// TwinCAT 3 PLC project Main
// ProgramVersion: 3.1.4023.0
// libraries:
//   mobject-collections, * (mobject)
//   mobject-enumerable, * (mobject)
//   mobject-events, * (mobject)
//   Tc2_System, * (Beckhoff Automation GmbH)
//   Tc3_Module, * (Beckhoff Automation GmbH)
//   TcUnit, * (www.tcunit.org)
// project tree:
//   / PlcTask.TcTTO
//   POUs/ Main.TcPOU
//   Tests/ OrderedDicKeyValueForwardEnumerator_TestSuite.TcPOU (not stored), OrderedDictionaryForwardEnumerator_TestSuite.TcPOU (not stored), DictionaryKeyValueForwardEnumerator_TestSuite.TcPOU (not stored), Dictionary_TestSuite.TcPOU (not stored), DictionaryForwardEnumerator_TestSuite.TcPOU (not stored), OrderedDictionary_TestSuite.TcPOU (not stored), LinkedList_TestSuite.TcPOU (not stored), ListForwardEnumerator_TestSuite.TcPOU, List_TestSuite.TcPOU, StackForwardEnumerator_TestSuite.TcPOU (not stored), Queue_TestSuite.TcPOU (not stored), LinkedListForwardEnumerator_TestSuite.TcPOU (not stored), Stack_TestSuite.TcPOU (not stored), QueueForwardEnumerator_TestSuite.TcPOU (not stored)
//   Tests/Mocks/EventHandlers/ CollectionChangedEventHandler.TcPOU (not stored), CollectionDisposedEventHandler.TcPOU (not stored), CollectionEventHandler.TcPOU (not stored), KeyValueCollectionChangedEventHandler.TcPOU (not stored), KeyValueCollectionEventHandler.TcPOU (not stored), KeyValueCollectionDisposedEventHandler.TcPOU (not stored), MockEventHandler.TcPOU (not stored)
// real-time tasks:
//   TASK PlcTask: cycle T#10ms, priority 20, ADS port 350

CONFIGURATION Main
    RESOURCE PLC ON TwinCAT3
        TASK PlcTask(INTERVAL := T#10ms, PRIORITY := 20);
        PROGRAM Main WITH PlcTask : Main;
    END_RESOURCE
END_CONFIGURATION

// ---- POUs/Main.TcPOU
PROGRAM Main
VAR
	dictionary_TestSuite : Dictionary_TestSuite;
	dictionaryForwardEnumerator_TestSuite : DictionaryForwardEnumerator_TestSuite;
	dictionaryKeyValueForwardEnumerator_TestSuite : DictionaryKeyValueForwardEnumerator_TestSuite;
	orderedDictionary_TestSuite : OrderedDictionary_TestSuite;
	orderedDictionaryForwardEnumerator_TestSuite : OrderedDictionaryForwardEnumerator_TestSuite;
	orderedDicKeyValueForwardEnumerator_TestSuite : OrderedDicKeyValueForwardEnumerator_TestSuite;
    linkedList_TestSuite : LinkedList_TestSuite;
	linkedListForwardEnumerator_TestSuite : LinkedListForwardEnumerator_TestSuite;
    list_TestSuite : List_TestSuite;
    listEnumerator_TestSuite : ListForwardEnumerator_TestSuite;
	queue_TestSuite : Queue_TestSuite;
	queueForwardEnumerator_TestSuite : QueueForwardEnumerator_TestSuite;
    stack_TestSuite : Stack_TestSuite;
	stackForwardEnumerator_TestSuite : StackForwardEnumerator_TestSuite;
END_VAR

TcUnit.Run();

END_PROGRAM

// ---- Tests/List_TestSuite.TcPOU
FUNCTION_BLOCK List_TestSuite EXTENDS TcUnit.FB_TestSuite
VAR
END_VAR

CheckAddItem();
CheckCapacityAfterAdding1Item();
CheckCapacityAfterAdding5Items();
CheckCapacityAfterAdding5ItemsTrimThen1Item();
CheckCapacityAtStart();
CheckClear();
CheckContains();
CheckTryCopyTo();
CheckTryCopyToLocation();
CheckCount();
CheckGetByIndexInBounds();
CheckGetByIndexNoItems();
CheckGetByIndexOutOfBounds();
CheckGetEnumerator();
CheckGetIndexOfExistingItem();
CheckGetIndexOfNonExistingItem();
CheckImplementsICollection();
CheckImplementsIList();
CheckTryInsert();
CheckOnChangedEvent();
CheckOnDisposedEvent();
CheckOnceEvent();
CheckOffEvent();
CheckTryRemoveAtInBounds();
CheckTryRemoveAtNoItems();
CheckTryRemoveAtOutOfBounds();
CheckTryRemoveItemFirstShiftUp();
CheckTryRemoveItemNonExisting();
CheckTryRemoveItemSecondShiftUp();
CheckTrimExcessAfterAdding5Items();
CheckIsEmptyWhenEmpty();
CheckIsEmptyWhenFull();

METHOD PRIVATE CheckAddItem
VAR
	in1 : INT := 123;
	in2 : INT := 456;
	in3 : INT := 789;
	out : INT;
	expected : INT := 789;
END_VAR
VAR_INST
	list : List;
END_VAR
TEST('CheckAddItem');

list.AddItem(in1); // [123]
list.AddItem(in2); // [123,456]
list.AddItem(in3); // [123,456,789]

list.TryGetByIndex(2, out);

AssertEquals(expected, out, 'Did not produce the expected result');

TEST_FINISHED();
END_METHOD

METHOD PRIVATE CheckCapacityAfterAdding1Item
VAR
	in1 : INT := 1;
	expected : DINT := 4;
	out : DINT;
END_VAR
VAR_INST
	list : List;
END_VAR
TEST('CheckCapacityAfterAdding1Item');

list.AddItem(in1); // [1, null, null, null]

out := list.Capacity;

AssertEquals(expected, out, 'List was expected to double once 5 items were added');

TEST_FINISHED();
END_METHOD

METHOD PRIVATE CheckCapacityAfterAdding5Items
VAR
	in1 : INT := 1;
	in2 : INT := 2;
	in3 : INT := 3;
	in4 : INT := 4;
	in5 : INT := 5;
	in6 : INT := 6;
	expected : DINT := 8;
	out : DINT;
END_VAR
VAR_INST
	list : List;
END_VAR
TEST('CheckCapacityAfterAdding5Items');

list.AddItem(in1); // [1, null, null, null]
list.AddItem(in2); // [1, 2, null, null]
list.AddItem(in3); // [1, 2, 3, null]
list.AddItem(in4); // [1, 2, 3, 4]
list.AddItem(in5); // [1, 2, 3, 4, 5, null, null, null]

out := list.Capacity;

AssertEquals(expected, out, 'List was expected to double once 5 items were added');

TEST_FINISHED();
END_METHOD

METHOD PRIVATE CheckCapacityAfterAdding5ItemsTrimThen1Item
VAR
	in1 : INT := 1;
	in2 : INT := 2;
	in3 : INT := 3;
	in4 : INT := 4;
	in5 : INT := 5;
	in6 : INT := 6;
	expected : DINT := 10;
	out : DINT;
END_VAR
VAR_INST
	list : List;
END_VAR
TEST('CheckCapacityAfterAdding5ItemsTrimThen1Item');

list.AddItem(in1); // [1, null, null, null]
list.AddItem(in2); // [1, 2, null, null]
list.AddItem(in3); // [1, 2, 3, null]
list.AddItem(in4); // [1, 2, 3, 4]
list.AddItem(in5); // [1, 2, 3, 4, 5, null, null, null]
list.TrimExcess(); // [1, 2, 3, 4, 5]
list.AddItem(in6); // [1, 2, 3, 4, 5, 6]

out := list.Capacity;

AssertEquals(expected, out, 'Incorrect capacity returned');

TEST_FINISHED();
END_METHOD

METHOD PRIVATE CheckCapacityAtStart
VAR
	expected : DINT := 0;
	out : DINT;
END_VAR
VAR_INST
	list : List;
END_VAR
TEST('CheckCapacityAtStart');

out := list.Capacity;

AssertEquals(expected, out, 'List was expected to start with a capacity of 0');

TEST_FINISHED();
END_METHOD

METHOD PRIVATE CheckClear
VAR
	in1 : INT := 123;
	in2 : INT := 456;
	in3 : INT := 789;
	expected : INT := 789;
	out : INT;
END_VAR
VAR_INST
	list : List;
END_VAR
TEST('CheckClear');

list.AddItem(in1); // [123]
list.AddItem(in2); // [123,456]

list.Clear(); // []
list.AddItem(in3); // [789]

list.TryGetByIndex(0, out);

AssertEquals(expected, out, 'Did not produce the expected result');

TEST_FINISHED();
END_METHOD

METHOD PRIVATE CheckContains
VAR
	in1 : INT := 123;
	in2 : INT := 456;
	in3 : INT := 789;
	result : BOOL;
END_VAR
VAR_INST
	list : List;
END_VAR
TEST('ListTests_CheckContains');

list.AddItem(in1); // [123]
list.AddItem(in2); // [123,456]
list.AddItem(in3); // [123,456,789]

result := list.Contains(in2);

AssertTrue(result, 'Contains returned false while item should be in collection');

TEST_FINISHED();
END_METHOD

METHOD PRIVATE CheckCount
VAR
	in1 : INT := 123;
	in2 : INT := 456;
	in3 : INT := 789;
	expected : DINT := 3;
	out : DINT;
END_VAR
VAR_INST
	list : List;
END_VAR
TEST('ListTests_CheckCount');

list.AddItem(in1); // [123]
list.AddItem(in2); // [123,456]
list.AddItem(in3); // [123,456,789]

out := list.Count;

AssertEquals(expected, out, 'Did not prodocue the expected result');

TEST_FINISHED();
END_METHOD

METHOD PRIVATE CheckGetByIndexInBounds
VAR
	in1 : INT := 123;
	in2 : INT := 456;
	in3 : INT := 789;
	out : INT;
	result : BOOL;
	expected : INT := 456;
END_VAR
VAR_INST
	list : List;
END_VAR
TEST('CheckGetByIndexInBounds');

list.AddItem(in1); // [123]
list.AddItem(in2); // [123,456]
list.AddItem(in3); // [123,456,789]

result := list.TryGetByIndex(1, out);

AssertTRUE(result, 'Returned FALSE while the index is populated');

AssertEquals(expected, out, 'Retrieved different value than expected');

TEST_FINISHED();
END_METHOD

METHOD PRIVATE CheckGetByIndexNoItems
VAR
	out : INT;
	result : BOOL;
END_VAR
VAR_INST
	list : List;
END_VAR
TEST('CheckGetByIndexNoItems');

result := list.TryGetByIndex(0, out);

AssertFalse(result, 'Returned TRUE while no items exist');

TEST_FINISHED();
END_METHOD

METHOD PRIVATE CheckGetByIndexOutOfBounds
VAR
	in1 : INT := 123;
	in2 : INT := 456;
	in3 : INT := 789;
	out : INT;
	result : BOOL;
END_VAR
VAR_INST
	list : List;
END_VAR
TEST('ListTests_CheckGetByIndexOutOfBounds_ReturnsFalse');

list.AddItem(in1); // [123]
list.AddItem(in2); // [123,456]
list.AddItem(in3); // [123,456,789]

result := list.TryGetByIndex(3, out);

AssertFalse(result, 'Returned TRUE while the index is not populated');

TEST_FINISHED();
END_METHOD

METHOD PRIVATE CheckGetEnumerator
VAR
	in1 : INT := 123;
	in2 : INT := 456;
	in3 : INT := 789;
	enumerator : I_ForwardEnumerator;
	result : BOOL;
END_VAR
VAR_INST
	list : List;
END_VAR
TEST('CheckGetEnumerator');

list.AddItem(in1); // [123]
list.AddItem(in2); // [123,456]
list.AddItem(in3); // [123,456,789]

enumerator := list.GetEnumerator();

AssertTrue(
	Condition := (enumerator <> 0),
	Message := 'Did not return an enumerator'
);

enumerator.Dispose();

TEST_FINISHED();
END_METHOD

METHOD PRIVATE CheckGetIndexOfExistingItem
VAR
	in1 : INT := 123;
	in2 : INT := 456;
	in3 : INT := 789;
	expected : DINT := 1;
	result : DINT;
END_VAR
VAR_INST
	list : List;
END_VAR
TEST('CheckGetIndexOfExistingItem');

list.AddItem(in1); // [123]
list.AddItem(in2); // [123,456]
list.AddItem(in3); // [123,456,789]

result := list.GetIndexOf(in2);

AssertEquals(result, expected, 'The index is not the expected index');

TEST_FINISHED();
END_METHOD

METHOD PRIVATE CheckGetIndexOfNonExistingItem
VAR
	in1 : INT := 123;
	in2 : INT := 456;
	in3 : INT := 789;
	expected : DINT := -1;
	result : DINT;
END_VAR
VAR_INST
	list : List;
END_VAR
TEST('CheckGetIndexOfNonExistingItem');

list.AddItem(in1); // [123]
list.AddItem(in2); // [123,456]

result := list.GetIndexOf(in3);

AssertEquals(result, expected, 'The index is not -1 which indicates missing');

TEST_FINISHED();
END_METHOD

METHOD PRIVATE CheckImplementsICollection
VAR
    collection : I_Collection := list;
    result : BOOL;
END_VAR
VAR_INST
	list : List;
END_VAR
TEST('ListTests_CheckImplementsICollection');

result := collection <> 0;

AssertTrue(result, 'Did not implement ICollection');

TEST_FINISHED();
END_METHOD

METHOD PRIVATE CheckImplementsIEnumerable
VAR
	enumerable : I_Enumerable := list;
	result : BOOL;
END_VAR
VAR_INST
	list : List;
END_VAR
TEST('CheckImplementsIEnumerable');

result := enumerable <> 0;

AssertTrue(result, 'Did not implement IEnumerable');

TEST_FINISHED();
END_METHOD

METHOD PRIVATE CheckImplementsIList
VAR
    iList : I_List := list;
    result : BOOL;
END_VAR
VAR_INST
	list : List;
END_VAR
TEST('ListTests_CheckImplementsIList');

result := iList <> 0;

AssertTrue(Condition := result,
    Message := 'Did not implement IList');

TEST_FINISHED();
END_METHOD

METHOD PUBLIC CheckIsEmptyWhenEmpty
VAR
	result : BOOL;
END_VAR
VAR_INST
	list : List;
END_VAR
TEST('CheckIsEmptyWhenEmpty');

// @TEST-RUN
result := list.IsEmpty;

// @TEST-ASSSERT
AssertTrue(
	Condition := result,
	Message := 'Incorrect state of IsEmpty'
);

TEST_FINISHED();
END_METHOD

METHOD PUBLIC CheckIsEmptyWhenFull
VAR
	in : INT := 123;
	result : BOOL;
END_VAR
VAR_INST
	list : List;
END_VAR
TEST('CheckIsEmptyWhenFull');

// @TEST-FIXTURE
list.AddItem(in);

// @TEST-RUN
result := list.IsEmpty;

// @TEST-ASSSERT
AssertFalse(
	Condition := result,
	Message := 'Incorrect state of IsEmpty'
);

TEST_FINISHED();
END_METHOD

METHOD PUBLIC CheckOffEvent
VAR
	value : INT := 123;
	handler : CollectionChangedEventHandler(ExpectedOriginator := list);
END_VAR
VAR_INST
	list : List;
END_VAR
TEST('CheckOffEvent');

// @TEST-FIXTURE
list.OnEvent('OnChanged',handler);
list.OffEvent('OnChanged',handler);

// @TEST-RUN
list.AddItem(value);

// @TEST-ASSSERT
AssertFalse(
	Condition := handler.EventReceived,
	Message := 'OnceEvent emitted the OnChanged event more than once'
);

TEST_FINISHED();
END_METHOD

METHOD PUBLIC CheckOnceEvent
VAR
	value : INT := 123;
	handler : CollectionChangedEventHandler(ExpectedOriginator := list);
END_VAR
VAR_INST
	list : List;
END_VAR
TEST('CheckOnceEvent');

// @TEST-FIXTURE
list.OnceEvent('OnChanged',handler);
list.AddItem(value);
handler.Reset();

// @TEST-RUN
list.AddItem(value);

// @TEST-ASSSERT
AssertFalse(
	Condition := handler.EventReceived,
	Message := 'OnceEvent emitted the OnChanged event more than once'
);

TEST_FINISHED();
END_METHOD

METHOD PUBLIC CheckOnChangedEvent
VAR
	value : INT := 123;
	handler : CollectionChangedEventHandler(ExpectedOriginator := list);
END_VAR
VAR_INST
	list : List;
END_VAR
TEST('CheckOnChangedEvent');

// @TEST-FIXTURE
list.OnEvent('OnChanged',handler);

// @TEST-RUN
list.AddItem(value);

// @TEST-ASSSERT
AssertTrue(
	Condition := handler.EventReceived,
	Message := 'Did not emit the OnChanged event'
);

AssertTrue(
	Condition := handler.FromExpectedOriginator,
	Message := 'Did not include itself in the OnChanged event'
);

TEST_FINISHED();
END_METHOD

METHOD PUBLIC CheckOnDisposedEvent
VAR
	pList : POINTER TO List;
	handler : CollectionDisposedEventHandler(ExpectedOriginator := 0);
END_VAR
TEST('CheckOnDisposedEvent');

// @TEST-FIXTURE
pList := __NEW(List);
handler.SetExpectedOriginator(pList^);
pList^.OnEvent('OnDisposed',handler);

// @TEST-RUN
pList^.Dispose();

// @TEST-ASSSERT
AssertTrue(
	Condition := handler.EventReceived,
	Message := 'Did not emit the OnDisposed event'
);

AssertTrue(
	Condition := handler.FromExpectedOriginator,
	Message := 'Did not include itself in the OnDisposed event'
);

TEST_FINISHED();
END_METHOD

METHOD PRIVATE CheckTrimExcessAfterAdding5Items
VAR
	in1 : INT := 1;
	in2 : INT := 2;
	in3 : INT := 3;
	in4 : INT := 4;
	in5 : INT := 5;
	in6 : INT := 6;
	expected : DINT := 5;
	out : DINT;
END_VAR
VAR_INST
	list : List;
END_VAR
TEST('CheckTrimExcessAfterAdding5Items');

list.AddItem(in1); // [1, null, null, null]
list.AddItem(in2); // [1, 2, null, null]
list.AddItem(in3); // [1, 2, 3, null]
list.AddItem(in4); // [1, 2, 3, 4]
list.AddItem(in5); // [1, 2, 3, 4, 5, null, null, null]
list.TrimExcess(); // [1, 2, 3, 4, 5]

out := list.Capacity;

AssertEquals(expected, out, 'List was expected to double once 5 items were added');

TEST_FINISHED();
END_METHOD

METHOD PRIVATE CheckTryCopyTo
VAR
	in1 : INT := 123;
	in2 : INT := 456;
	in3 : INT := 789;
	out : ARRAY [0..2] OF INT;
	expected : ARRAY [0..2] OF INT := [123,456,789];
END_VAR
VAR_INST
	list : List;
END_VAR
TEST('CheckTryCopyTo');

list.AddItem(in1); // [123]
list.AddItem(in2); // [123,456]
list.AddItem(in3); // [123,456,789]

list.TryCopyTo(out);

AssertEquals(
	Expected := expected,
	Actual := out,
	Message := 'Did not produce the expected result'
);

TEST_FINISHED();
END_METHOD

METHOD PRIVATE CheckTryCopyToLocation
VAR
	in1 : INT := 123;
	in2 : INT := 456;
	in3 : INT := 789;
	out : ARRAY [0..2] OF INT;
	expected : ARRAY [0..2] OF INT := [123,456,789];
END_VAR
VAR_INST
	list : List;
END_VAR
TEST('CheckTryCopyToLocation');

list.AddItem(in1); // [123]
list.AddItem(in2); // [123,456]
list.AddItem(in3); // [123,456,789]

list.TryCopyToLocation(ADR(out),SIZEOF(out));

AssertEquals(
	Expected := expected,
	Actual := out,
	Message := 'Did not produce the expected result'
);

TEST_FINISHED();
END_METHOD

METHOD PRIVATE CheckTryInsert
VAR
	in1 : INT := 123;
	in2 : INT := 456;
	in3 : INT := 789;
	out : INT;
	result : BOOL;
	expected : INT := 789;
END_VAR
VAR_INST
	list : List;
END_VAR
TEST('CheckTryInsert');

list.AddItem(in1); // [123]
list.AddItem(in1); // [123,456]
list.TryInsert(1, in3); // [123,789,456]

list.TryGetByIndex(1,out);

AssertEquals(expected, out, 'Did not produce the expected result');

TEST_FINISHED();
END_METHOD

METHOD PRIVATE CheckTryRemoveAtInBounds
VAR
	in1 : INT := 123;
	in2 : INT := 456;
	in3 : INT := 789;
	out : INT;
	result : BOOL;
END_VAR
VAR_INST
	list : List;
END_VAR
TEST('CheckTryRemoveAtInBounds');

list.AddItem(in1); // [123]
list.AddItem(in2); // [123,456]
list.AddItem(in3); // [123,456,789]

list.TryRemoveAt(0);

result := list.TryGetByIndex(0, out);

AssertTrue(result, 'Couldnt get first item');
AssertEquals(in2, out, 'Array didnt shift up items');

TEST_FINISHED();
END_METHOD

METHOD PRIVATE CheckTryRemoveAtNoItems
VAR
	out : INT;
	result : BOOL;
END_VAR
VAR_INST
	list : List;
END_VAR
TEST('CheckTryRemoveAtNoItems');

result := list.TryRemoveAt(0);

AssertFalse(result, 'Returned true while there was nothing to remove');

TEST_FINISHED();
END_METHOD

METHOD PRIVATE CheckTryRemoveAtOutOfBounds
VAR
	in1 : INT := 123;
	in2 : INT := 456;
	in3 : INT := 789;
	out : INT;
	result : BOOL;
END_VAR
VAR_INST
	list : List;
END_VAR
TEST('CheckTryRemoveAtOutOfBounds');

list.AddItem(in1); // [123]
list.AddItem(in2); // [123,456]
list.AddItem(in3); // [123,456,789]

result := list.TryRemoveAt(3);

AssertFalse(result, 'Returned true while remove was out of bounds');

TEST_FINISHED();
END_METHOD

METHOD PRIVATE CheckTryRemoveItemFirstShiftUp
VAR
	in1 : INT := 123;
	in2 : INT := 456;
	in3 : INT := 789;
	out : INT;
	result : BOOL;
	expected : INT := 456;
END_VAR
VAR_INST
	list : List;
END_VAR
TEST('CheckTryRemoveItemFirstShiftUp');

list.AddItem(in1); // [123]
list.AddItem(in2); // [123,456]
list.AddItem(in3); // [123,456,789]
list.TryRemoveItem(in1); // [456,789]

result := list.TryGetByIndex(0, out);

AssertTrue(result, 'Couldnt get first item');

AssertEquals(expected, out, 'Array didnt shift up items');

TEST_FINISHED();
END_METHOD

METHOD PRIVATE CheckTryRemoveItemNonExisting
VAR
	in1 : INT := 123;
	in2 : INT := 456;
	in3 : INT := 789;
	out : INT;
	result : BOOL;
END_VAR
VAR_INST
	list : List;
END_VAR
TEST('CheckTryRemoveItemNonExisting');

list.AddItem(in1); // [123]
list.AddItem(in2); // [123,456]

result := list.TryRemoveItem(in3);

AssertFalse(result, 'RemoveItem returned true which should not happen when item does not exist');

TEST_FINISHED();
END_METHOD

METHOD PRIVATE CheckTryRemoveItemSecondShiftUp
VAR
	in1 : INT := 123;
	in2 : INT := 456;
	in3 : INT := 789;
	out : INT;
	result : BOOL;
	expected : INT := 789;
END_VAR
VAR_INST
	list : List;
END_VAR
TEST('CheckTryRemoveItemSecondShiftUp');

list.AddItem(in1); // [123]
list.AddItem(in2); // [123,456]
list.AddItem(in3); // [123,456,789]
list.TryRemoveItem(in2); // [123,789]

result := list.TryGetByIndex(1, out);

AssertTrue(result, 'Coulndt get first item');
AssertEquals(expected, out, 'Array didnt shift up items');

TEST_FINISHED();
END_METHOD

END_FUNCTION_BLOCK

// ---- Tests/ListForwardEnumerator_TestSuite.TcPOU
FUNCTION_BLOCK ListForwardEnumerator_TestSuite EXTENDS TcUnit.FB_TestSuite
VAR
END_VAR

CheckIsValidAtStart();
CheckMoveNextReturnsFalseAtTheEnd();
CheckMoveNextReturnsTrueSingleItem();
CheckMoveNextReturnsFalseWhenEmpty();
CheckMoveNextReturnsTrueMultipleItems();
CheckReset();
CheckTryGet();
CheckTryGetTo();
CheckWorksWithArrays();
CheckWorksWithIntegers();
CheckWorksWithStrings();

METHOD PRIVATE CheckIsValidAtStart
VAR
	result : BOOL;
	enumerator : I_ForwardEnumerator;
END_VAR
VAR_INST
	store : List;
END_VAR
TEST('CheckIsValidAtStart');

enumerator := store.GetEnumerator();

result := enumerator.IsValid;
enumerator.Dispose();

AssertTrue(
	Condition := result,
	Message := 'IsValid returned false'
);

TEST_FINISHED();
END_METHOD

METHOD PRIVATE CheckMoveNextReturnsFalseAtTheEnd
VAR
	in1 : INT := 123;
	result : BOOL;
	enumerator : I_ForwardEnumerator;
END_VAR
VAR_INST
	store : List;
END_VAR
TEST('CheckMoveNextReturnsFalseAtTheEnd');

store.AddItem(in1);
enumerator := store.GetEnumerator();

enumerator.MoveNext();
result := enumerator.MoveNext();
enumerator.Dispose();

AssertFalse(result,
    'MoveNext did not correctly signal the end of the enumeration');
	
TEST_FINISHED();
END_METHOD

METHOD PRIVATE CheckMoveNextReturnsFalseWhenEmpty
VAR
	result : BOOL;
	enumerator : I_ForwardEnumerator;
	count : DINT;
END_VAR
VAR_INST
	store : List;
END_VAR
TEST('CheckMoveNextReturnsFalseWhenEmpty');

count := store.Count;
enumerator := store.GetEnumerator();

result := enumerator.MoveNext();
enumerator.Dispose();

AssertFalse(Condition := result,
    Message := 'MoveNext did not correctly signal the end of the enumeration');

TEST_FINISHED();
END_METHOD

METHOD PRIVATE CheckMoveNextReturnsTrueMultipleItems
VAR
	in1 : INT := 123;
	in2 : INT := 456;
	in3 : INT := 789;
	result : BOOL;
	enumerator : I_ForwardEnumerator;
END_VAR
VAR_INST
	store : List;
END_VAR
TEST('CheckMoveNextReturnsTrueMultipleItems');

store.AddItem(in1);
store.AddItem(in2);
store.AddItem(in3);
enumerator := store.GetEnumerator();

result := enumerator.MoveNext();
enumerator.Dispose();

AssertTrue(result, 'MoveNext did not correctly signal there were more items to follow');

TEST_FINISHED();
END_METHOD

METHOD PRIVATE CheckMoveNextReturnsTrueSingleItem
VAR
	in1 : INT := 123;
	result : BOOL;
	enumerator : I_ForwardEnumerator;
END_VAR
VAR_INST
	store : List;
END_VAR
TEST('CheckMoveNextReturnsTrueSingleItem');

store.AddItem(in1);
enumerator := store.GetEnumerator();

result := enumerator.MoveNext();
enumerator.Dispose();

AssertTrue(result,
    'MoveNext did not correctly signal there were more items to follow');
	
TEST_FINISHED();
END_METHOD

METHOD PRIVATE CheckReset
VAR
	in1 : ARRAY [0..1] OF REAL := [0.1,2.3];
	in2 : ARRAY [0..1] OF REAL := [1.2,3.4];
	in3 : ARRAY [0..1] OF REAL := [2.3,4.5];
	out : ARRAY [0..1] OF REAL;
	expected : ARRAY [0..1] OF REAL := [0.1,2.3];
	enumerator : I_ForwardEnumerator;
END_VAR
VAR_INST
	store : List;
END_VAR
TEST('CheckReset');

store.AddItem(in1);
store.AddItem(in2);
store.AddItem(in3);

enumerator := store.GetEnumerator();

enumerator.MoveNext();
enumerator.MoveNext();
enumerator.Reset();
enumerator.MoveNext();
enumerator.TryGet(out);

enumerator.Dispose();

AssertEquals(
	Expected := expected,
	Actual := out,
	Message := 'Did not produce the expected result'
);

TEST_FINISHED();
END_METHOD

METHOD PRIVATE CheckTryGet
VAR
	in : INT := 123;
	out : INT;
	expected : INT := 123;
	result : BOOL;
	enumerator : I_ForwardEnumerator;
END_VAR
VAR_INST
	store : List;
END_VAR
TEST('CheckTryGet');

store.AddItem(in);
enumerator := store.GetEnumerator();
enumerator.MoveNext();

result := enumerator.TryGet(out);
enumerator.Dispose();

AssertTrue(
	Condition := result,
	Message := 'Method returned false'
);

AssertEquals(
	Expected := expected,
	Actual := out,
	Message := 'Did not produce the expected result'
);

TEST_FINISHED();
END_METHOD

METHOD PRIVATE CheckTryGetTo
VAR
	in : INT := 123;
	out : INT;
	expected : INT := 123;
	result : BOOL;
	enumerator : I_ForwardEnumerator;
END_VAR
VAR_INST
	store : List;
END_VAR
TEST('CheckTryGetTo');

store.AddItem(in);
enumerator := store.GetEnumerator();
enumerator.MoveNext();

result := enumerator.TryGetTo(ADR(out),SIZEOF(out));
enumerator.Dispose();

AssertTrue(
	Condition := result,
	Message := 'Method returned false'
);

AssertEquals(
	Expected := expected,
	Actual := out,
	Message := 'Did not produce the expected result'
);

TEST_FINISHED();
END_METHOD

METHOD PRIVATE CheckWorksWithArrays
VAR
	in1 : ARRAY [0..1] OF REAL := [0.1,2.3];
	in2 : ARRAY [0..1] OF REAL := [1.2,3.4];
	in3 : ARRAY [0..1] OF REAL := [2.3,4.5];
	out1 : ARRAY [0..1] OF REAL;
	out2 : ARRAY [0..1] OF REAL;
	out3 : ARRAY [0..1] OF REAL;
	expected1 : ARRAY [0..1] OF REAL := [0.1,2.3];
	expected2 : ARRAY [0..1] OF REAL := [1.2,3.4];
	expected3 : ARRAY [0..1] OF REAL := [2.3,4.5];
	enumerator : I_ForwardEnumerator;
END_VAR
VAR_INST
	store : List;
END_VAR
TEST('CheckWorksWithArrays');

store.AddItem(in1);
store.AddItem(in2);
store.AddItem(in3);

enumerator := store.GetEnumerator();

enumerator.MoveNext();
enumerator.TryGet(out1);
enumerator.MoveNext();
enumerator.TryGet(out2);
enumerator.MoveNext();
enumerator.TryGet(out3);

enumerator.Dispose();

AssertEquals(
	Expected := expected1,
	Actual := out1,
	Message := 'Did not produce the expected 1st result'
);

AssertEquals(
	Expected := expected2,
	Actual := out2,
	Message := 'Did not produce the expected 2nd result'
);

AssertEquals(
	Expected := expected3,
	Actual := out3,
	Message := 'Did not produce the expected 3rd result'
);

TEST_FINISHED();
END_METHOD

METHOD PRIVATE CheckWorksWithIntegers
VAR
	in1 : INT := 123;
	in2 : INT := 234;
	in3 : INT := 345;
	out1 : INT;
	out2 : INT;
	out3 : INT;
	expected1 : INT := 123;
	expected2 : INT := 234;
	expected3 : INT := 345;
	enumerator : I_ForwardEnumerator;
END_VAR
VAR_INST
	store : List;
END_VAR
TEST('CheckWorksWithIntegers');

store.AddItem(in1);
store.AddItem(in2);
store.AddItem(in3);

enumerator := store.GetEnumerator();

enumerator.MoveNext();
enumerator.TryGet(out1);
enumerator.MoveNext();
enumerator.TryGet(out2);
enumerator.MoveNext();
enumerator.TryGet(out3);

enumerator.Dispose();

AssertEquals(
	Expected := expected1,
	Actual := out1,
	Message := 'Did not produce the expected 1st result'
);

AssertEquals(
	Expected := expected2,
	Actual := out2,
	Message := 'Did not produce the expected 2nd result'
);

AssertEquals(
	Expected := expected3,
	Actual := out3,
	Message := 'Did not produce the expected 3rd result'
);

TEST_FINISHED();
END_METHOD

METHOD PRIVATE CheckWorksWithStrings
VAR
	in1 : STRING := 'test1';
	in2 : STRING := 'test2';
	in3 : STRING := 'test3';
	out1 : STRING;
	out2 : STRING;
	out3 : STRING;
	expected1 : STRING := 'test1';
	expected2 : STRING := 'test2';
	expected3 : STRING := 'test3';
	enumerator : I_ForwardEnumerator;
END_VAR
VAR_INST
	store : List;
END_VAR
TEST('CheckWorksWithStrings');

store.AddItem(in1);
store.AddItem(in2);
store.AddItem(in3);

enumerator := store.GetEnumerator();

enumerator.MoveNext();
enumerator.TryGet(out1);
enumerator.MoveNext();
enumerator.TryGet(out2);
enumerator.MoveNext();
enumerator.TryGet(out3);

enumerator.Dispose();

AssertEquals(
	Expected := expected1,
	Actual := out1,
	Message := 'Did not produce the expected 1st result'
);

AssertEquals(
	Expected := expected2,
	Actual := out2,
	Message := 'Did not produce the expected 2nd result'
);

AssertEquals(
	Expected := expected3,
	Actual := out3,
	Message := 'Did not produce the expected 3rd result'
);

TEST_FINISHED();
END_METHOD

END_FUNCTION_BLOCK
